{attribute 'linkalways'} 
{attribute 'no_explicit_call' := 'This FB is a CLASS and must be accessed using methods or properties'}
{attribute 'enable_dynamic_creation'}
FUNCTION_BLOCK _Array0To7OfByte EXTENDS ArrayDatatypeBase_1D
VAR CONSTANT
	lBound : DINT := 0;
	uBound : DINT := 7;
END_VAR
VAR
	localData : ARRAY [lBound..uBound] OF BYTE;
	activeData : REFERENCE TO ARRAY [lBound..uBound] OF BYTE REF= localData;
	elements : ARRAY [lBound..uBound] OF _BYTE(0);
	baseType : _BYTE(0);
END_VAR

PROPERTY PUBLIC Address : PVOID
GET
Address := ADR(activeData);
END_GET
END_PROPERTY

PROPERTY PUBLIC BaseDatatype : I_Datatype
GET
BaseDatatype := baseType;
END_GET
END_PROPERTY

METHOD PUBLIC ClearReference
VAR_INPUT
END_VAR
activeData REF= localData;
SetElementReference();
END_METHOD

METHOD PUBLIC Clone : I_Datatype
VAR
    pClone : POINTER TO _Array0To7OfByte;
END_VAR
pClone := __NEW(_Array0To7OfByte());
pClone^.Value := Value;
Clone := pClone^;
END_METHOD

METHOD FB_init : BOOL
VAR_INPUT
	bInitRetains : BOOL; // if TRUE, the retain variables are initialized (warm start / cold start)
	bInCopyCode : BOOL;  // if TRUE, the instance afterwards gets moved into the copy code (online change)
END_VAR
SetElementReference();
END_METHOD

METHOD PUBLIC MakeReferenceTo
VAR_INPUT
	ReferenceTarget : REFERENCE TO ARRAY [lBound..uBound] OF BYTE;
END_VAR
activeData REF= ReferenceTarget;
SetElementReference();
END_METHOD

METHOD PROTECTED OnSerializeArrayValues
VAR_INPUT
	Serializer : I_Serializer;
END_VAR
VAR
	i : DINT;
END_VAR
FOR i := lBound TO uBound DO
	elements[i].SerializeWith(Serializer);
END_FOR
END_METHOD

METHOD PROTECTED SetElementReference
VAR_INPUT
END_VAR
VAR
	i : DINT;
END_VAR
FOR i := lBound TO uBound DO
	elements[i].MakeReferenceTo(activeData[i]);
END_FOR
END_METHOD

PROPERTY PUBLIC Size : UDINT
GET
Size := SIZEOF(activeData);
END_GET
END_PROPERTY

METHOD PROTECTED TryDeserializeArrayValues : BOOL
VAR_INPUT
	Deserializer : I_Deserializer;
	Feedback : I_DeserializerFeedback;
END_VAR
VAR
	enumerator : I_DeserializerArrayForwardEnumerator;
	i : DINT;
END_VAR
enumerator := Deserializer.GetArrayEnumerator();
i := lBound;

WHILE enumerator.MoveNext() AND i <= uBound DO
	
	IF NOT elements[i].TryDeserializeFrom(enumerator.Current, Feedback) THEN
		EXIT;
	END_IF
	i := i + 1;

END_WHILE
enumerator.Dispose();
END_METHOD

METHOD PUBLIC TryGetElementAsDatatypeByIndex : BOOL
VAR_INPUT
	Index : DINT;
	Destination : REFERENCE TO I_Datatype;
END_VAR
IF Index < lbound OR Index > ubound THEN
	RETURN;
END_IF

Destination := elements[Index];
TryGetElementAsDatatypeByIndex := TRUE;
END_METHOD

METHOD PUBLIC TryGetLowerBound : BOOL
VAR_INPUT
	Dimention : UDINT;
	Destination : REFERENCE TO DINT;
END_VAR
IF Dimention = 1 THEN
	Destination := lBound;
	TryGetLowerBound := TRUE;
END_IF
END_METHOD

METHOD PUBLIC TryGetUpperBound : BOOL
VAR_INPUT
	Dimention : UDINT;
	Destination : REFERENCE TO DINT;
END_VAR
IF Dimention = 1 THEN
	Destination := uBound;
	TryGetUpperBound := TRUE;
END_IF
END_METHOD

METHOD TryMakeReferenceTo : BOOL
VAR_INPUT
	Target : I_Datatype;
END_VAR
VAR
	targetAsArray : I_ArrayDatatype;
	pTargetData : POINTER TO ARRAY [lBound..uBound] OF BYTE;
END_VAR
IF NOT Target.TryResolveAsArrayDatatype(targetAsArray) THEN
	RETURN;
END_IF

IF NOT (targetAsArray.Identifier = Identifier) THEN
	RETURN;
END_IF

pTargetData := Target.Address;
activeData REF= pTargetData^;
SetElementReference();
TryMakeReferenceTo := TRUE;
END_METHOD

PROPERTY PUBLIC Value : REFERENCE TO ARRAY [lBound..uBound] OF BYTE;
GET
Value ref= activeData;
END_GET
END_PROPERTY

END_FUNCTION_BLOCK

(* stored: Version 1.1.0.1, ProductVersion 3.1.4024.13
   POU _Array0To7OfByte: Id {34d6c557-707a-0ec3-18d1-bf2fd8013757}, SpecialFunc None
   Folder Core: Id {f259791f-81a2-03cf-154b-51c13a2b57f3}
   Folder Constructor: Id {23cbc157-abec-066f-1426-9ba50aa778e8}
   Folder Protected: Id {59cfb482-2376-00ba-21b3-0bc389581d9b}
   Folder Customize: Id {9f6e1f43-2f92-0a6b-2ff3-b561cdef770d}
   Property Address: Id {4d7249f0-433b-0a9c-2a56-546e0569a845}
   Get Get: Id {e55008f6-1c3a-0cad-0af9-11149d314c0e}
   Property BaseDatatype: Id {ae873d56-fbc3-075d-15b8-38f866a044d1}
   Get Get: Id {021aaf93-34e6-0862-3022-8660f06a0ae7}
   Method ClearReference: Id {ab5414ba-bd50-06f4-23af-6a3f9c920b34}
   Method Clone: Id {352ce499-a261-04b9-2966-12ecbce3599a}
   Method FB_init: Id {a02504a0-5339-08b8-319d-c4611b3713f0}
   Method MakeReferenceTo: Id {585232a2-8012-0a33-050b-e6ffac9c98fb}
   Method OnSerializeArrayValues: Id {db98b889-5bff-0c9b-25ba-ed0c64e8787f}
   Method SetElementReference: Id {718dcd0d-6277-0a37-0499-c46675fe5c30}
   Property Size: Id {cf9e3126-a852-0301-3c61-d32b601f7196}
   Get Get: Id {4b666d0a-5154-0ecc-1073-41f5ebdc1036}
   Method TryDeserializeArrayValues: Id {d2772691-4a38-0579-00f5-e827ca20957a}
   Method TryGetElementAsDatatypeByIndex: Id {7f34354c-72c3-04a7-3649-fb0c9e8b4c0e}
   Method TryGetLowerBound: Id {a906ef8e-1044-0377-1749-c2d9da3d4354}
   Method TryGetUpperBound: Id {213f1f3a-8b85-04f4-2498-6f882246a55f}
   Method TryMakeReferenceTo: Id {8118a94a-d581-0df5-1c91-af9dc17d8c7c}
   Property Value: Id {d5d66595-f118-07c4-1422-0f7c568b089f}
   Get Get: Id {d52e9d41-d6cc-01e4-245e-e2655019da15} *)
